{attribute 'qualified_only'}
VAR_GLOBAL
	StateProteza : UDINT;
	StateCurrentProteza : DINT;
	BoolProteza  : BOOL := TRUE;
END_VAR

(* stored: Version 1.1.0.1
   GVL GVL: Id {e704112c-6181-0958-0436-a320982b8db1} *)
